{attribute addProperty BoxType "EKM1101-0000-0016"}
{attribute addProperty Id "StatusAT %I*Status_BD85E94F162"}
{attribute addProperty CRC "3947416948"}
{attribute addProperty SizeInBites "16"}
{attribute addProperty SizeInBytes "2"}
TYPE MMS_Device_Inputs_EB48CD74 :
STRUCT
	{attribute addProperty Name "Status"}
	Status AT %I* : Status_BD85E94F;
END_STRUCT
END_TYPE

(* stored: Version 1.2.0.0, ProductVersion 3.1.4024.9
   DUT MMS_Device_Inputs_EB48CD74: Id {57e3fa62-a2ae-4e42-a32f-6a1990bbfe54} *)
